FUNCTION_BLOCK TestType
  (* Version 1.0, 2005-04-08, Goran Cengic, Chalmers *)
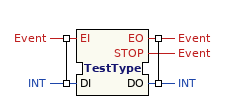
  EVENT_INPUT
    EI WITH DI;
  END_EVENT
  EVENT_OUTPUT
    EO WITH DO;
    STOP;
  END_EVENT
  VAR_INPUT
    DI : INT;
  END_VAR
  VAR_OUTPUT
    DO : INT;
  END_VAR
  VAR
    invoked : INT;
  END_VAR
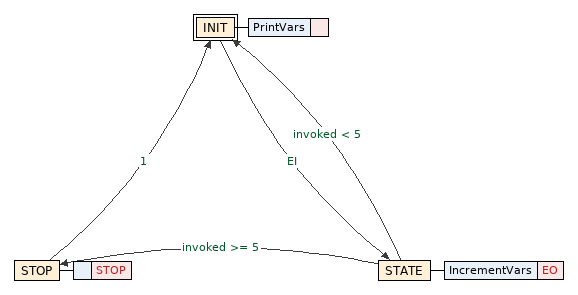
  EC_STATES
    INIT : PrintVars;
    STATE : IncrementVars -> EO;
    STOP : -> STOP;
  END_STATES
  EC_TRANSITIONS
    INIT TO STATE := EI;
    STATE TO INIT := invoked < 5;
    STATE TO STOP := invoked >= 5;
    STOP TO INIT := 1;
  END_TRANSITIONS
  ALGORITHM IncrementVars IN Java:
      invoked = invoked + 1;
      DO = DI + 1;
  END_ALGORITHM
  ALGORITHM PrintVars IN Java:
      System.out.println("invoked: " + invoked);
      System.out.println("DO: " + DO);
  END_ALGORITHM
END_FUNCTION_BLOCK
